PROGRAM LogicandCountersex01
VAR
	S1				: DigitalInput_NO;
	P1				: DigitalOutput;
	CV				: INT  := 0;
	S1_flank		: R_trig;
END_VAR

S1_flank(clk := S1.isOn);

IF S1_flank.Q THEN
	CV := CV + 1;
END_IF

IF CV >= 5 THEN
	P1.On();
END_IF

END_PROGRAM

(* stored: Version 1.1.0.1
   POU LogicandCountersex01: Id {764718b6-b938-4406-84b0-98fdd54b7b80}, SpecialFunc None *)
